// TwinCAT 3 PLC project PLC
// ProgramVersion: 3.1.4026.19
// CompilerDefines: VISU_USEPROPERTYINFO
// libraries:
//   SPT Base Types, * (Beckhoff Automation LLC)
//   SPT Components, * (Beckhoff Automation LLC)
//   SPT Diagnostic, * (Beckhoff Automation LLC)
//   SPT EtherCat, * (Beckhoff Automation LLC)
//   SPT Event Logger, * (Beckhoff Automation LLC)
//   SPT Motion Control, * (Beckhoff Automation LLC)
//   SPT Utilities, * (Beckhoff Automation LLC)
//   Tc2_Standard, * (Beckhoff Automation GmbH)
//   Tc2_System, * (Beckhoff Automation GmbH)
//   Tc3_EventLogger, * (Beckhoff Automation GmbH)
//   Tc3_PackML_V3, * (Beckhoff Automation GmbH)
// project tree:
//   / GlobalTextList.TcGTLO, PlcTask.TcTTO, Visualization Manager.TcVMO (not stored)
//   GVLs/ GVL_Axes.TcGVL
//   Modules/00 Machine/DUTs/ ST_Machine_Cfg.TcDUT, ST_Machine_Cmd.TcDUT, ST_Machine_HMI.TcDUT, ST_Machine_Sts.TcDUT
//   Modules/00 Machine/ Machine.TcPOU
//   Modules/01 Press/ Press.TcPOU
//   POUs/ MAIN.TcPOU
//   VISUs/ Visualization.TcVIS
// real-time tasks:
//   TASK PlcTask: cycle T#10ms, priority 20, ADS port 350
// motion (NC):
//   TASK NC-Task 1 SAF: cycle T#2ms, priority 4, ADS port 501
//   TASK NC-Task 1 SVB: cycle T#10ms, priority 8, ADS port 511
//   AXIS Axis 1 (id 1)
//   AXIS Axis 2 (id 2)
//   AXIS Axis 3 (id 3)
//   AXIS Axis 4 (id 4)
//   AXIS Axis 5 (id 5)
//   AXIS Axis 6 (id 6)
//     OtherSettings: AllowMotionCmdToSlave=true
//     encoder EncType=1
//     drive DrvType=5
//       Analog: TorqueSetpointScale=10, ScaleFactorActTorque=0.1
//     controller CtrType=1
//       CtrPara: PriorControlFactor=1
//         Observer: BandWidth=20
//   AXIS Axis 7 (id 7)
//     OtherSettings: AllowMotionCmdToSlave=true
//     encoder EncType=1
//     drive DrvType=5
//       Analog: TorqueSetpointScale=10, ScaleFactorActTorque=0.1
//     controller CtrType=1
//       CtrPara: PriorControlFactor=1
//         Observer: BandWidth=20
//   AXIS Axis 8 (id 8)
//     OtherSettings: AllowMotionCmdToSlave=true
//     encoder EncType=1
//     drive DrvType=5
//       Analog: TorqueSetpointScale=10, ScaleFactorActTorque=0.1
//     controller CtrType=1
//       CtrPara: PriorControlFactor=1
//         Observer: BandWidth=20
//   AXIS Axis 9 (id 9)
//     OtherSettings: AllowMotionCmdToSlave=true
//     encoder EncType=1
//     drive DrvType=5
//       Analog: TorqueSetpointScale=10, ScaleFactorActTorque=0.1
//     controller CtrType=1
//       CtrPara: PriorControlFactor=1
//         Observer: BandWidth=20
//   AXIS Axis 10 (id 10)
//     OtherSettings: AllowMotionCmdToSlave=true
//     encoder EncType=1
//     drive DrvType=5
//       Analog: TorqueSetpointScale=10, ScaleFactorActTorque=0.1
//     controller CtrType=1
//       CtrPara: PriorControlFactor=1
//         Observer: BandWidth=20
// variable links:
//   PLC/PLC Instance <-> NC-Task 1 SAF/Axes/Axis 1
//     PlcTask Inputs/GVL_Axes.Axis[1].BasicAxis._Axis.NcToPlc <-> Outputs/ToPlc
//     PlcTask Outputs/GVL_Axes.Axis[1].BasicAxis._Axis.PlcToNc <-> Inputs/FromPlc
//   PLC/PLC Instance <-> NC-Task 1 SAF/Axes/Axis 10
//     PlcTask Inputs/GVL_Axes.Axis[10].BasicAxis._Axis.NcToPlc <-> Outputs/ToPlc
//     PlcTask Outputs/GVL_Axes.Axis[10].BasicAxis._Axis.PlcToNc <-> Inputs/FromPlc
//   PLC/PLC Instance <-> NC-Task 1 SAF/Axes/Axis 2
//     PlcTask Inputs/GVL_Axes.Axis[2].BasicAxis._Axis.NcToPlc <-> Outputs/ToPlc
//     PlcTask Outputs/GVL_Axes.Axis[2].BasicAxis._Axis.PlcToNc <-> Inputs/FromPlc
//   PLC/PLC Instance <-> NC-Task 1 SAF/Axes/Axis 3
//     PlcTask Inputs/GVL_Axes.Axis[3].BasicAxis._Axis.NcToPlc <-> Outputs/ToPlc
//     PlcTask Outputs/GVL_Axes.Axis[3].BasicAxis._Axis.PlcToNc <-> Inputs/FromPlc
//   PLC/PLC Instance <-> NC-Task 1 SAF/Axes/Axis 4
//     PlcTask Inputs/GVL_Axes.Axis[4].BasicAxis._Axis.NcToPlc <-> Outputs/ToPlc
//     PlcTask Outputs/GVL_Axes.Axis[4].BasicAxis._Axis.PlcToNc <-> Inputs/FromPlc
//   PLC/PLC Instance <-> NC-Task 1 SAF/Axes/Axis 5
//     PlcTask Inputs/GVL_Axes.Axis[5].BasicAxis._Axis.NcToPlc <-> Outputs/ToPlc
//     PlcTask Outputs/GVL_Axes.Axis[5].BasicAxis._Axis.PlcToNc <-> Inputs/FromPlc
//   PLC/PLC Instance <-> NC-Task 1 SAF/Axes/Axis 6
//     PlcTask Inputs/GVL_Axes.Axis[6].BasicAxis._Axis.NcToPlc <-> Outputs/ToPlc
//     PlcTask Outputs/GVL_Axes.Axis[6].BasicAxis._Axis.PlcToNc <-> Inputs/FromPlc
//   PLC/PLC Instance <-> NC-Task 1 SAF/Axes/Axis 7
//     PlcTask Inputs/GVL_Axes.Axis[7].BasicAxis._Axis.NcToPlc <-> Outputs/ToPlc
//     PlcTask Outputs/GVL_Axes.Axis[7].BasicAxis._Axis.PlcToNc <-> Inputs/FromPlc
//   PLC/PLC Instance <-> NC-Task 1 SAF/Axes/Axis 8
//     PlcTask Inputs/GVL_Axes.Axis[8].BasicAxis._Axis.NcToPlc <-> Outputs/ToPlc
//     PlcTask Outputs/GVL_Axes.Axis[8].BasicAxis._Axis.PlcToNc <-> Inputs/FromPlc
//   PLC/PLC Instance <-> NC-Task 1 SAF/Axes/Axis 9
//     PlcTask Inputs/GVL_Axes.Axis[9].BasicAxis._Axis.NcToPlc <-> Outputs/ToPlc
//     PlcTask Outputs/GVL_Axes.Axis[9].BasicAxis._Axis.PlcToNc <-> Inputs/FromPlc

CONFIGURATION PLC
    RESOURCE PLC ON TwinCAT3
        TASK PlcTask(INTERVAL := T#10ms, PRIORITY := 20);
        PROGRAM MAIN WITH PlcTask : MAIN;
    END_RESOURCE
END_CONFIGURATION

// ---- Modules/00 Machine/DUTs/ST_Machine_Cfg.TcDUT
TYPE ST_Machine_Cfg :
	STRUCT
	END_STRUCT
END_TYPE

// ---- Modules/00 Machine/DUTs/ST_Machine_Cmd.TcDUT
TYPE ST_Machine_Cmd :
	STRUCT
		MoveAll : BOOL;
	END_STRUCT
END_TYPE

// ---- Modules/00 Machine/DUTs/ST_Machine_HMI.TcDUT
TYPE ST_Machine_HMI :
	STRUCT
		Cmd : ST_Machine_Cmd;
		Cfg : ST_Machine_Cfg;
		Sts : ST_Machine_Sts;
	END_STRUCT
END_TYPE

// ---- Modules/00 Machine/DUTs/ST_Machine_Sts.TcDUT
TYPE ST_Machine_Sts :
	STRUCT
	END_STRUCT
END_TYPE

// ---- GVLs/GVL_Axes.TcGVL
{attribute 'qualified_only'}
VAR_GLOBAL
	// 1. Axes available for control by EMs
	Axis : ARRAY[1..MAX_AXES] OF FB_Component_BasicAxis;
END_VAR

VAR_GLOBAL CONSTANT
	MAX_AXES : INT := 10;
END_VAR

// ---- POUs/MAIN.TcPOU
PROGRAM MAIN
VAR
	Machine : Machine := (Name := 'Machine');
END_VAR

// All sample code provided by Beckhoff Automation LLC are for illustrative purposes only and are provided “as is” and without any warranties, express or implied. Actual implementations in applications will vary significantly. Beckhoff Automation LLC shall have no liability for, and does not waive any rights in relation to, any code samples that it provides or the use of such code samples for any purpose.

(*
	This sample code shows how an axis component can be dynamically (re)assigned to an Equipment Module.
	1. The axis components are declared as global variables.
	2. Each Equipment Module that will have access to the axis components has an array of interfaces of type I_BasicAxis.
		This interface will be used for accessing the methods and properties of the axis.
	3. A local instance I_ComponentBase is assigned using QueryInterface.
		This interface will be used to register the axis component with the Equipment Module.
	4. The Press Equipment Module has a VAR_INPUT for GroupID that is assigned when the EM is declared in Machine
			LeftPress  : Press := (Name := 'Left Press', GroupID := 0);
			RightPress : Press := (Name := 'Right Press', GroupID := 1);
	5. The Press.Initialize method registers the proper axis components to the Press EM
		a. Each GVL_Axes.Axis is assigned to the local _ipGlobalAxes array
		b. Using __QueryInterface each _ipGlobalAxes is cast to its _ipComponent interface
		c. If the _iAxisActive is equal to the GroupID, then the Component is registered to the EM
			Note: Initially the _iAxisActive array will be all 0s, and the GroupId for the Left Press is also 0
	6. After the first Initialization is complete all axes are now components of the LeftPress EM
	7. When the state machine of a Press EM reaches the Clearing state, all of the components are cleared and reassigned as configured
		a. _InitComplete is set to FALSE and the ipComponents array is set to 0
			This will cause the Initialize method to be run again the next time CyclicLogic is called.
			With the ipComponents array filled with 0s all components will be registered again.
		b. When processing the Initialize method this time it is important that the _iAxisActive array now holds the GroupId that each axis should be assigned to.
		c. It is required that the SUPER^.Clearing method not be called until after the Initialization has been completed, otherwise a page fault will occur.
			To protect from this the SUPER^.Clearing method is called only when the _InitComplete is TRUE
		d. Because we are processing both the Initialize and the Clearing methods at the same time we must be aware of the hazard for parallel use of the (Descendent)SequenceState
			variable. Normally this is not a concern, but the Initialize method in the base class is using the SequenceState variable,
			and the Initialize method of the Press EM is using the DescendentSequenceState variable. 
			Therefore, if we were to use either of these in Clearing then we would create a condition where the two CASE statements are both modifying the value of the CASE 
			selection variable. As a remedy the variable ClearingState has been declared as a local variable in the Press EM. This variable is set to 0 in the Aborting method.  
	8. For this sample radio buttons have been added to a Visu that will allow each axis to be assigned to either the Left or Right Press EM.
		a. The radio buttons are assigned to the variable MAIN.Machine.AxisAssignment[X], where x is replaced by the Axis number to be assigned.
			Using a radio button ensures that an axis can only be assigned to a single EM.
			The radio buttons will write an INT value to the selected variable, in this situation the value written by the radio button matches with the GroupId
		b. In Machine.Clearing the ActiveAxes property of both LeftPress and RightPress are set to the AxisAssignment. This will pass the radio button selections to each EM.
		c. In the ActiveAxes.Set _iAxisActive is popluated with the data.
		d. Now when the Initialize method is run during Clearing, each axis will be assigned to an EM based on the selected radio button. 
	9. Enabling and Controlling the correct axes
		a. Commands for all axes can be accessed throught the _ipGlobalAxes array, however this can be dangerous and should not be done.
		b. An array of _ipLocalAxes is declared in the Press EM that will hold the address of the proper GLV_Axes.Axis for the EM.
		c. In the Initialize method the array of _ipLocalAxes is set to 0 along with the NumberOfLocalAxes
		d. When all checks have passed and a component is registerd the _ipLocalAxes[i] is assigned to the value of the _ipGlobalAxes[i],
			and the NumberOfLocalAxes is increased by 1. This ensures that the list of _ipLocalAxes only contains the addresses of the GVL_Axes that are controlled by this EM.
		e. In the Resetting method the axes are enabled. The FOR loop is from 1 to GVL_Axes.MAX_AXES and the code checks that the _ipLocalAxes[i] is not 0 before issuing a commnd.
	10. To operate this sample:
		a. Use the Visu to assign each axis to either the Left or Right Press EM.
		b. If not in the state Aborted, issue the Abort command with the Abort button
		c. Press the Clear button
			Once the state machine is in Stopped you can check the LeftPress or RightPress local variable declaration and expand the ipComponents array
			The number of indexes with values should match the number of axes configured in the Visu.
			If you expand an item in the array you will see the details of that item.
			Note: this array is different from the _ipComponent array that is used in the Initialize method for registering the components, that array should always be full.
		d. Continue to move the state machine to Execute
		e. Press the Move All button and the axes assigned to the Left Press will move forward by 100, and the axes assigned to the Right Press will be in Reverse by 100.
		f. Return to step 9a and repeat the process with a different axis configuration.	
			
*)

// For Debug Only
_AppInfo.KeepOutputsOnBP := TRUE;

//
Machine.CyclicLogic();

END_PROGRAM

// ---- Modules/00 Machine/Machine.TcPOU
FUNCTION_BLOCK Machine EXTENDS FB_PackML_BaseModule
VAR
	LeftPress  : Press := (Name := 'Left Press', GroupId := 0);	 //4. GroupId used to match up with AxisAssignment
	RightPress : Press := (Name := 'Right Press', GroupId := 1); //4. GroupId used to match up with AxisAssignment

	//
	AxisAssignment : ARRAY[1..GVL_AXES.MAX_AXES] OF INT;

	//
	HMI : ST_Machine_HMI;
END_VAR

(* This method contains code which will execute when this PackML module is in the Clearing state*)
METHOD PROTECTED Clearing
// 8.b. This will pass the radio button selections to each EM.
LeftPress.ActiveAxes  := AxisAssignment;
RightPress.ActiveAxes := AxisAssignment;

//
SUPER^.Clearing();
END_METHOD

METHOD CyclicLogic
IF NOT _InitComplete THEN
	_InitComplete := Initialize();
	RETURN;
END_IF

SUPER^.CyclicLogic();
END_METHOD

(* This method contains code which will execute when this PackML module is in the Execute state*)
METHOD PROTECTED Execute
CASE _CurrentMode OF
	E_PMLUnitMode.Production:
		IF HMI.Cmd.MoveAll THEN
			HMI.Cmd.MoveAll := FALSE;
			LeftPress.MoveAll(100.0);
			RightPress.MoveAll(-100.0);
		END_IF
END_CASE
END_METHOD

(* Automatically enables and disables HMI control based on the PackML mode*)
METHOD PROTECTED HMIPermissions
AllowHMIControl(TRUE);
END_METHOD

(* Basic module initialization logic*)
METHOD PROTECTED Initialize : BOOL
Initialize := FALSE;
CASE DescendantSequenceState OF
	0:
		RegisterSubmodule(SubModule := LeftPress);
		RegisterSubmodule(SubModule := RightPress);
		DescendantSequenceState := DescendantSequenceState + 10;

	10:
		IF SUPER^.Initialize() THEN
			DescendantSequenceState := DescendantSequenceState + 10;
		END_IF

	20:
		Initialize := TRUE;
END_CASE
END_METHOD

END_FUNCTION_BLOCK

// ---- Modules/01 Press/Press.TcPOU
FUNCTION_BLOCK Press EXTENDS FB_PackML_BaseModule
VAR_INPUT
	GroupId : USINT; //4. Assigned during declaration, used to match up with AxisAssignment
END_VAR

VAR
	_ipGlobalAxes	  : ARRAY[1..GVL_Axes.MAX_AXES] OF I_BasicAxis; // 2. Interface to be assigned to a Globally declared axis
	_iAxisActive	  : ARRAY[1..GVL_Axes.MAX_AXES] OF INT;
	_ipLocalAxes	  : ARRAY[1..GVL_Axes.MAX_AXES] OF I_BasicAxis; // 9.b. Hold the addresses of the active GLV_Axes.Axis for the EM
	NumberOfLocalAxes : INT;

	//
	ClearingState : INT; // 7.d
END_VAR

(* This method contains code which will execute when this PackML module is in the Aborting state*)
METHOD PROTECTED Aborting
ClearingState := 0; // 7.d.
SUPER^.Aborting();
END_METHOD

PROPERTY ActiveAxes : ARRAY[1..GVL_AXES.MAX_AXES] OF INT
GET
ActiveAxes := _iAxisActive;
END_GET
SET
_iAxisActive := ActiveAxes; // 8.c.
END_SET
END_PROPERTY

(* This method contains code which will execute when this PackML module is in the Clearing state*)
METHOD PROTECTED Clearing
VAR
	i : UDINT;
END_VAR
CASE ClearingState OF
	0:
		// 7.a. _InitComplete is set to FALSE and the ipComponents array is set to 0
		_InitComplete := FALSE;
		FOR i := 1 TO NumberOfComponents DO
			ipComponents[i] := 0;
		END_FOR

		ClearingState := ClearingState + 10;

	10:
		IF _InitComplete THEN
			ClearingState := ClearingState + 10;
		END_IF

	20:
		StateTasksComplete := TRUE;
END_CASE

// 7.c. It is required that the SUPER^.Clearing method not be called until after the Initialization has been completed, otherwise a page fault will occur.
IF _InitComplete THEN
	SUPER^.Clearing();
END_IF
END_METHOD

METHOD CyclicLogic
IF NOT _InitComplete THEN
	_InitComplete := Initialize();
	RETURN;
END_IF

SUPER^.CyclicLogic();
END_METHOD

(* Basic module initialization logic*)
METHOD PROTECTED Initialize : BOOL
VAR
	i			 : INT;
	_ipComponent : I_ComponentBase; // 3. Interface to be used for RegisterComponent
END_VAR
Initialize := FALSE;
CASE DescendantSequenceState OF
	0: // 5.a. Each GVL_Axes.Axis is assigned to the local _ipAxes array
		FOR i := 1 TO GVL_Axes.MAX_AXES DO
			_ipGlobalAxes[i] := GVL_Axes.Axis[i];
		END_FOR

		// 9.c. The list of _ipLocalAxis is cleared
		FOR i := 1 TO GVL_Axes.MAX_AXES DO
			_ipLocalAxes[i] := 0;
		END_FOR

		DescendantSequenceState := DescendantSequenceState + 10;

	10:
		NumberOfLocalAxes := 0; // 9.c. Set the count to 0
		FOR i := 1 TO GVL_Axes.MAX_AXES DO
			// 5.b. Using __QueryInterface each _ipAxis is cast to its _ipComponent interface
			IF __QUERYINTERFACE(_ipGlobalAxes[i], _ipComponent) THEN
				// 5.c. 7.b. 8.d. If the _iAxisActive is equal to the GroupID, then the Component is registered to the EM
				IF (_iAxisActive[i] = GroupId) THEN
					RegisterComponent(Component := _ipComponent);

					// 9.d. Copy the address from the Global to the Local to issue commands and check status of axes assigned to this EM only
					_ipLocalAxes[i]	  := _ipGlobalAxes[i];
					NumberOfLocalAxes := NumberOfLocalAxes + 1;
				END_IF
			END_IF
		END_FOR

		DescendantSequenceState := DescendantSequenceState + 10;

	20:
		IF SUPER^.Initialize() THEN
			DescendantSequenceState := DescendantSequenceState + 10;
		END_IF

	30:
		Initialize := TRUE;
END_CASE
END_METHOD

METHOD MoveAll : BOOL
VAR_INPUT
	Position : LREAL;
END_VAR

VAR
	i : INT;
END_VAR
MoveAll := FALSE;

//
FOR i := 1 TO GVL_Axes.MAX_AXES DO
	IF _ipLocalAxes[i] <> 0 THEN
		_ipLocalAxes[i].MoveRelative(Position, TRUE);
	END_IF
END_FOR

//

(*FOR i := 1 TO GVL_Axes.MAX_AXES DO
	IF (_iAxisActive[i] = GroupId) AND_THEN _ipAxes[i].MoveRelative(Position, TRUE) THEN
		;
	END_IF
END_FOR*)
END_METHOD

(* This method contains code which will execute when this PackML module is in the Resetting state*)
METHOD PROTECTED Resetting
VAR
	i	  : INT;
	count : INT;
END_VAR
CASE SequenceState OF
	0:
		NoStateTasksToComplete := FALSE;
		SequenceState		   := SequenceState + 10;

	10: // 9.e. Enable only the Locally controlled axes
		FOR i := 1 TO GVL_Axes.MAX_AXES DO
			IF _ipLocalAxes[i] <> 0 THEN
				_ipLocalAxes[i].Enable();
			END_IF
		END_FOR

		SequenceState := SequenceState + 10;

	20:
		count := 0;
		FOR i := 1 TO GVL_Axes.MAX_AXES DO
			// 9.e. loop through all axes, but only check the status of the locally controlled axes
			IF (_ipLocalAxes[i] <> 0) AND_THEN _ipLocalAxes[i].Enabled THEN
				count := count + 1;
			END_IF
		END_FOR

		IF (count = NumberOfLocalAxes) THEN
			SequenceState := SequenceState + 10;
		END_IF

	30:
		StateTasksComplete := TRUE;
END_CASE

SUPER^.Resetting();
END_METHOD

END_FUNCTION_BLOCK

// ---- GlobalTextList.TcGTLO
TEXTLIST GlobalTextList
  278 = 'Axis 1'
  381 = 'Axis 10'
  898 = 'Axis 2'
  421 = 'Axis 3'
  662 = 'Axis 4'
  402 = 'Axis 5'
  141 = 'Axis 6'
  682 = 'Axis 7'
  63 = 'Axis 8'
  192 = 'Axis 9'
  957 = 'Left'
  150 = 'Move All'
  164 = 'Right'
END_TEXTLIST

// ---- VISUs/Visualization.TcVIS
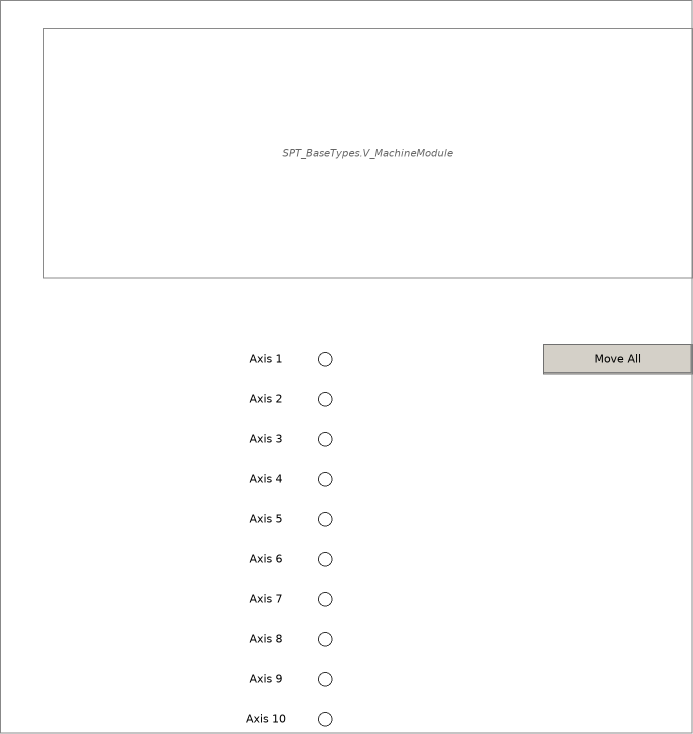
VISUALIZATION Visualization  // 693x734
    Frame (43,28 650x250)
        shows SPT_BaseTypes.V_MachineModule(HMI := MAIN.Machine.PackMLBaseModule_HMI)
    RadioButton (316,344 150x30), variable: MAIN.Machine.AxisAssignment[1]
        Areas[0]: Text=Left
        Areas[1]: Text=Right
    Label (226,344 80x30), "Axis 1"
    RadioButton (316,384 150x30), variable: MAIN.Machine.AxisAssignment[2]
        Areas[0]: Text=Left
        Areas[1]: Text=Right
    Label (226,384 80x30), "Axis 2"
    RadioButton (316,424 150x30), variable: MAIN.Machine.AxisAssignment[3]
        Areas[0]: Text=Left
        Areas[1]: Text=Right
    Label (226,424 80x30), "Axis 3"
    RadioButton (316,464 150x30), variable: MAIN.Machine.AxisAssignment[4]
        Areas[0]: Text=Left
        Areas[1]: Text=Right
    Label (226,464 80x30), "Axis 4"
    RadioButton (316,504 150x30), variable: MAIN.Machine.AxisAssignment[5]
        Areas[0]: Text=Left
        Areas[1]: Text=Right
    Label (226,504 80x30), "Axis 5"
    RadioButton (316,544 150x30), variable: MAIN.Machine.AxisAssignment[6]
        Areas[0]: Text=Left
        Areas[1]: Text=Right
    Label (226,544 80x30), "Axis 6"
    RadioButton (316,584 150x30), variable: MAIN.Machine.AxisAssignment[7]
        Areas[0]: Text=Left
        Areas[1]: Text=Right
    Label (226,584 80x30), "Axis 7"
    RadioButton (316,624 150x30), variable: MAIN.Machine.AxisAssignment[8]
        Areas[0]: Text=Left
        Areas[1]: Text=Right
    Label (226,624 80x30), "Axis 8"
    RadioButton (316,664 150x30), variable: MAIN.Machine.AxisAssignment[9]
        Areas[0]: Text=Left
        Areas[1]: Text=Right
    Label (226,664 80x30), "Axis 9"
    RadioButton (316,704 150x30), variable: MAIN.Machine.AxisAssignment[10]
        Areas[0]: Text=Left
        Areas[1]: Text=Right
    Label (226,704 80x30), "Axis 10"
    Button (543,344 150x30), "Move All"
        tap MAIN.Machine.HMI.Cmd.MoveAll
END_VISUALIZATION
